FUNCTION Clesious_to_faringate : REAL
VAR_INPUT
END_VAR
VAR
END_VAR

END_FUNCTION

(* stored: Version 1.1.0.1, ProductVersion 3.1.4024.12
   POU Clesious_to_faringate: Id {f2a1ad5d-45b7-4dd1-8149-2f30a871a48a}, SpecialFunc None *)
